TYPE E_InitializeState : (
    INIT_IDLE := 0,
    INIT_CLEAR_TRANSIENTS := 10,
    INIT_VALIDATE_MODE_SOURCE := 20,
    INIT_VALIDATE_COMMUNICATION := 30,
    INIT_VALIDATE_SENSORS := 40,
    INIT_RESET_AXIS_ERRORS := 50,
    INIT_HOME_Z_IF_REQUIRED := 60,
    INIT_HOME_R_IF_REQUIRED := 70,
    INIT_STOP_R := 80,
    INIT_RETURN_Z_REFERENCE := 90,
    INIT_RETURN_CYLINDERS := 100,
    INIT_RESET_FEEDER := 110,
    INIT_VALIDATE_CALIBRATIONS := 120,
    INIT_VALIDATE_ACTIVE_PROGRAM := 130,
    INIT_FINAL_READY_CHECK := 140,
    INIT_COMPLETE := 150,
    INIT_FAILED := 200
); END_TYPE

(* stored: Version 1.1.0.1
   DUT E_InitializeState: Id {E3000000-0000-4000-8000-000000000004} *)
